// TIA Portal V17 export
// export: Created 2025-06-26T06:49:25.8574839Z, ExportSetting WithDefaults, DisplayName Totally Integrated Automation Portal, DisplayVersion V17 Update 8, DisplayName TIA Portal Openness, DisplayVersion V17 Update 8, DisplayName TIA Portal Version Control Interface, DisplayVersion V17, DisplayName STEP 7 Professional, DisplayVersion V17 Update 8, DisplayName STEP 7 Safety, DisplayVersion V17 Update 6, DisplayName WinCC Advanced, DisplayVersion V17 Update 8
DATA_BLOCK "DB_State"   // DB12
{ S7_Optimized_Access := 'TRUE' }
AUTHOR : Heaten
VERSION : 0.1
// stored: AutoNumber true, DBAccessibleFromOPCUA true, DBAccessibleFromWebserver true, IsOnlyStoredInLoadMemory false, IsRetainMemResEnabled false, IsWriteProtectedInAS false, MemoryReserve 100
   VAR
      SystemInitialised : Bool;
      StopRequired : Bool;
      FastStop : Bool;
      StopLock : Bool;   // Not used
      ForceStateChangeFlags : Array[1..16] of Bool;
      RunningConditions : Struct
         ShaftSealSystemOK : Bool;
         OilHeatOK : Bool;
         HeatSinkTemperatureOK : Bool;
         HeatSourceTemperatureOK : Bool;
         SuperheatCompressorInOK : Bool;
         PressureSpreadOK : Bool;
         SuperheatCompressorOutOK : Bool;
         RecuperatorWorking : Bool;
         AtOrAboveHydrolockSpeed : Bool;
         SuctionLineDry : Bool;
         AuxiliariesOK : Bool;
         HeatSourceFlowOK : Bool;
         HeatSinkFlowOK : Bool;
         LubricationPrimingOk : Bool;
         DoWarmStart : Bool;
         CompressorStopped : Bool;
         RiskOfHydrolock : Bool;
      END_STRUCT;
      State : Struct
         State_Number : Int := -1;
         "0_Initialisation" : Bool;
         "1_Offline" : Bool;
         "2_Standby" : Bool;
         "3_PrepareStart" : Bool;
         "4_Start" : Bool;
         "5_Warmup" : Bool;
         "6_Running" : Bool;
         "7_Stop" : Bool;
      END_STRUCT;
      StatePauseFlags { S7_SetPoint := 'True'} : Array[0..7] of Bool;   // Allow pausing (level signal)
      StateConfirmFlags : Array[0..7] of Bool;   // Confirm past pause (momentary signal)
      StateDwellTimeElapsed : Array[0..8] of Bool;
   END_VAR
BEGIN
END_DATA_BLOCK
